Yaskawa INFORM job: R1_W27-A4(90,180)KM-OK.JBI

/JOB
//NAME R1_W27-A4(90,180)KM-OK
///FOLDERNAME KRIS-SCIANA
//POS
///NPOS 187,187,0,9,0,0
///TOOL 0
///POSTYPE PULSE
///PULSE
C00000=12408,-168229,-129239,-11856,76417,-1490
C00001=114075,-55562,-33330,-57879,69757,-51049
C00002=170127,-11218,4712,-80761,69619,-75034
C00003=166026,1115,14662,-80935,66751,-75417
C00004=166026,1115,14662,-80935,66751,-75417
C00005=164179,6139,17196,-85884,73779,-76491
C00006=163843,5639,16762,-85908,73539,-76507
C00007=164179,6139,17196,-85884,73779,-76491
C00008=166496,-467,13337,-75702,58764,-75189
C00009=166831,-1552,12436,-75705,58996,-75152
C00010=166508,-36,14521,-75997,58636,-74926
C00011=166831,-1552,12436,-75705,58996,-75152
C00012=166496,-467,13337,-75702,58764,-75189
C00013=166021,-3570,934,-78534,68009,-78358
C00014=137610,-28929,-19421,-69080,47942,-64710
C00015=100776,-35686,-23013,-57930,21837,-49720
C00016=103071,-36442,-26491,-56591,24205,-50318
C00017=97018,-28630,-27379,-22144,28331,-59500
C00018=96837,-21698,-21046,-22140,27966,-59499
C00019=100662,-29228,-19206,-55793,22319,-50751
C00020=102053,-30601,-20713,-56706,23278,-50281
C00021=94369,-26080,-26288,-14236,29524,-61616
C00022=90809,-41559,-31122,-11258,24098,-63096
C00023=90635,-42168,-31044,-11137,23721,-63156
C00024=94073,-53021,-44279,-15136,26788,-61156
C00025=105496,-45084,-28829,-64380,24182,-46446
C00026=105496,-45084,-28829,-64380,-61448,-46446
C00027=120732,-139011,-128731,-13191,-67324,37746
C00028=120732,-139011,-128731,-13191,-67324,37746
C00029=15630,-139011,-128731,-13191,-67324,37746
C00030=37783,65902,-41793,-18959,93512,79890
C00031=21816,-138429,-128213,-9073,25992,35710
C00032=3312,-138429,-128213,-9073,25992,35710
C00033=8567,85289,-13174,2735,78610,-10465
C00034=97991,22164,19578,-1121,74303,-36101
C00035=113962,41790,17661,4351,37010,-36101
C00036=153447,-77745,-45385,11807,63175,6285
C00037=169394,-84609,-38838,16107,56709,15659
C00038=173881,-75690,-28267,15647,54036,17014
C00039=174396,-73921,-25835,15662,53377,17117
C00040=174409,-72642,-23726,15788,52756,17025
C00041=174396,-73921,-25835,15662,53377,17117
C00042=177237,-69247,-20992,27235,53512,13633
C00043=177890,-67562,-19632,27129,53343,13864
C00044=177237,-69247,-20992,27235,53512,13633
C00045=181977,-77418,-24251,27266,50136,14704
C00046=193956,-50227,-14941,-539,58562,29056
C00047=192915,-50819,-15265,-329,58451,28665
C00048=194756,-48721,-14111,-700,58831,29355
C00049=182531,-71466,-31778,1788,58094,24759
C00050=122199,17749,55230,64618,69888,-3761
C00051=124469,25360,65490,65961,67496,-4502
C00052=125352,28797,70143,66592,66515,-4877
C00053=125200,39134,82378,67427,65683,-5911
C00054=125978,39297,82548,67654,65232,-5820
C00055=125200,39134,82378,67427,65683,-5911
C00056=125352,28797,70143,66592,66515,-4877
C00057=127676,20892,69191,78285,59026,-9362
C00058=127562,25294,74286,78756,58894,-9826
C00059=127676,21375,69995,78428,58968,-9490
C00060=125009,20842,69444,77518,60577,-9664
C00061=122672,36678,78518,58027,73309,-3381
C00062=122677,38905,82216,58303,72687,-3837
C00063=122672,36678,78518,58027,73309,-3381
C00064=169394,-84609,-38838,16107,56709,15659
C00065=192177,-39033,-19160,299,85673,46850
C00066=192177,-34142,-7713,300,81140,46844
C00067=191273,-36033,-8917,230,80912,46543
C00068=190571,-37450,-9806,174,80732,46307
C00069=191000,-36591,-9270,208,80842,46449
C00070=191000,-37231,-10676,208,81378,46450
C00071=190373,-38486,-11456,158,81216,46242
C00072=190373,-38091,-10592,158,80886,46242
C00073=190373,-40536,-16053,159,82992,46244
C00074=118612,15198,38856,55022,83195,1057
C00075=133487,-1087,21013,35992,98849,64323
C00076=137132,-5726,26455,36615,92702,63739
C00077=137287,-7082,25375,36660,92613,63770
C00078=137132,-5726,26455,36615,92702,63739
C00079=137132,-4574,28724,36576,92049,63519
C00080=137132,-5726,26455,36615,92702,63739
C00081=135105,9364,31394,36359,97356,64485
C00082=137553,-19599,1652,32898,84560,61916
C00083=145396,-31747,-6442,33707,80478,63803
C00084=146058,-32230,-6758,33764,80175,63976
C00085=145396,-31747,-6442,33707,80478,63803
C00086=145396,-32381,-7876,33664,80944,63945
C00087=145635,-34810,-9443,33705,80615,63940
C00088=145635,-34478,-8700,33728,80373,63868
C00089=145635,-34810,-9443,33705,80615,63940
C00090=166958,-28260,-6522,34091,73535,70390
C00091=170921,-25100,-2173,34137,71094,71258
C00092=171490,-25282,-2297,34116,70859,71419
C00093=170921,-25100,-2173,34137,71094,71258
C00094=170921,-25785,-3769,34024,71622,71427
C00095=171866,-27898,-5215,34016,71085,71649
C00096=171866,-27525,-4348,34079,70800,71557
C00097=171866,-27898,-5215,34016,71085,71649
C00098=170413,-50683,-19184,37966,51947,77320
C00099=172186,-18361,1190,35695,54496,79271
C00100=175964,-9154,13477,35828,50627,79612
C00101=176352,-9219,13425,35709,50467,79746
C00102=175964,-9154,13477,35828,50627,79612
C00103=175964,-10038,11459,35461,51274,79877
C00104=176713,-11464,10718,35354,50747,80043
C00105=176713,-11144,11450,35487,50511,79947
C00106=176713,-11464,10718,35354,50747,80043
C00107=123076,-83185,-29574,44713,66004,60586
C00108=132807,-78951,-22653,44198,75112,68451
C00109=133029,-79369,-22050,44355,74587,68307
C00110=133442,-81220,-22681,44553,73994,68215
C00111=133280,-79395,-22588,44357,74706,68467
C00112=133284,-82173,-24950,44353,74724,68477
C00113=133854,-84143,-25057,44659,73784,68294
C00114=133789,-83559,-24494,44652,73780,68264
C00115=133789,-82965,-23605,44700,73605,68182
C00116=133789,-83559,-24494,44652,73780,68264
C00117=126764,-78223,-26799,42400,79954,67989
C00118=129779,-124310,-39885,59101,44128,50595
C00119=142359,-111009,-28991,70365,32429,46878
C00120=144435,-110863,-28981,70591,31368,47293
C00121=166637,-108168,-28907,68791,20141,53479
C00122=165685,-116661,-37003,67388,20889,53934
C00123=169317,-97643,-42504,39636,61921,25134
C00124=181806,-47831,-14195,30226,94440,40482
C00125=192217,-74733,-34955,23643,74815,40848
C00126=189039,-36338,-14362,23914,80418,40542
C00127=179036,-43494,-16720,35248,78492,35239
C00128=184921,-32781,-12708,31409,62196,49986
C00129=184567,-29470,-5587,32219,59878,49253
C00130=185969,-1035,16805,31607,54976,48516
C00131=184454,-6788,8530,31302,57322,48585
C00132=186295,-45172,-18023,32156,53759,48198
C00133=187719,-75788,-33082,34439,47747,46698
C00134=196206,-71365,-30868,20961,47500,52163
C00135=191632,-40680,-12057,24621,48037,49834
C00136=186300,-39428,-14940,31590,54648,48556
C00137=172329,-61780,-29172,35843,57798,43133
C00138=136853,-81161,-37735,39391,69197,31515
C00139=139314,-24647,17192,44556,110664,42025
C00140=134198,-53539,2603,44314,98424,40161
C00141=147007,-50232,4151,49976,93054,43060
C00142=144010,-50727,1445,48871,95437,42954
C00143=139156,-48548,-22547,50335,108120,47151
C00144=122197,265,20116,61362,75919,1585
C00145=148312,-18266,18073,35868,41105,22148
C00146=148389,-10811,27499,37215,39474,21366
C00147=148139,-7130,31782,37859,38978,20950
C00148=149047,-9416,30148,37653,38478,21229
C00149=148550,-6621,33826,38481,38019,20665
C00150=151250,-3570,34403,36506,37914,22272
C00151=150396,-8469,29288,36370,38763,22201
C00152=150383,-15985,19712,34952,40435,23027
C00153=136141,-317,34070,49048,57432,19039
C00154=137229,7022,44527,50381,55121,18205
C00155=137621,10190,48745,50908,54295,17886
C00156=137107,11277,51332,51470,53891,17317
C00157=136657,9562,48504,50983,54669,17581
C00158=137398,10846,49256,50891,54423,17845
C00159=137247,10896,49257,50876,54513,17818
C00160=136822,13685,51719,50910,54678,17683
C00161=136799,9316,46568,50416,55288,18069
C00162=135467,4556,38210,49073,57743,18855
C00163=136137,-10257,13643,45943,62583,21899
C00164=136139,-13457,6254,44950,64655,-57340
C00165=140525,19486,41917,27486,58532,-69458
C00166=158575,-22743,-5640,261,63822,-52267
C00167=201270,-72526,-20170,-41599,43995,-22865
C00168=208523,-61328,-5512,-45049,45103,-18922
C00169=210983,-54521,-945,-44398,50079,-19814
C00170=208926,-60351,-4855,-45020,45353,-18846
C00171=208139,-60468,-3279,-45679,44265,-18612
C00172=209884,-54474,-922,-44345,49597,-20126
C00173=202908,-51930,157,-43430,46646,-22304
C00174=208516,-61339,-5515,-45051,45097,-18922
C00175=207445,-70087,-17224,-43111,46602,-20424
C00176=181249,-65588,-30997,1667,65478,-39835
C00177=185098,-71138,-35276,1207,65193,-38466
C00178=182759,-75971,-40143,1483,65742,61063
C00179=206355,-41348,-16857,-5174,86104,67834
C00180=205860,-39116,-9742,-5254,82857,67803
C00181=199217,-16106,8750,-10349,89886,65622
C00182=195049,-32120,-9942,-6453,85783,64063
C00183=178413,-64785,-35080,-8104,82994,58638
C00184=153142,-115476,-42163,-24127,19724,-41141
C00185=118343,-192417,-136241,31416,17665,-73466
C00186=12522,-192417,-136241,31416,17665,-73466
BC00000=5573,1179356,685508
BC00001=17842,1187216,744485
BC00002=145005,1191142,773938
BC00003=169645,1191142,773938
BC00004=169645,1191142,773938
BC00005=170825,1191142,715041
BC00006=170825,1191142,715041
BC00007=170825,1191142,715041
BC00008=193098,1191142,831231
BC00009=203526,1191142,830949
BC00010=203526,1191142,830949
BC00011=203526,1191142,830949
BC00012=193098,1191142,831231
BC00013=169645,1191142,773938
BC00014=112075,1191142,777374
BC00015=47018,1191142,781257
BC00016=50087,1191142,764866
BC00017=51351,1191141,771759
BC00018=51351,1191141,771759
BC00019=51315,1191142,758310
BC00020=51315,1191142,758310
BC00021=51315,1191142,758310
BC00022=51315,1191142,758310
BC00023=51315,1191142,758310
BC00024=51315,1191142,758310
BC00025=47056,1191142,794711
BC00026=20889,1191142,794711
BC00027=33296,1190075,947302
BC00028=33296,691954,947302
BC00029=33296,691954,947302
BC00030=150689,509,1059807
BC00031=165933,1190075,1065356
BC00032=165933,1346249,1065356
BC00033=73688,729726,969252
BC00034=389559,778302,1060448
BC00035=389559,1189504,1060448
BC00036=393628,1104806,555119
BC00037=394257,1091704,476953
BC00038=399035,1282079,493083
BC00039=399035,1280810,493083
BC00040=399035,1280810,493083
BC00041=399035,1280810,493083
BC00042=399035,1261438,493083
BC00043=399035,1261313,493083
BC00044=399035,1261438,493083
BC00045=399035,1261438,493083
BC00046=399035,1290178,493083
BC00047=399035,1288101,493083
BC00048=399035,1290178,493083
BC00049=399035,1296613,493602
BC00050=399035,1384690,493083
BC00051=399035,1384690,493083
BC00052=399035,1384690,493083
BC00053=399035,1382924,493083
BC00054=399035,1382921,493083
BC00055=399035,1382924,493083
BC00056=399035,1384690,493083
BC00057=399035,1384690,493083
BC00058=399035,1384690,493083
BC00059=399035,1384690,493083
BC00060=399035,1384690,493083
BC00061=399035,1366830,493083
BC00062=399035,1367204,493083
BC00063=399035,1366830,493083
BC00064=394257,1091704,476953
BC00065=394257,1091704,476953
BC00066=394257,1091704,476953
BC00067=394257,1091704,476953
BC00068=394257,1091704,476953
BC00069=394257,1091704,476953
BC00070=394257,1091704,476953
BC00071=394257,1091704,476953
BC00072=394257,1091704,476953
BC00073=394257,1091704,476953
BC00074=394257,1176346,476953
BC00075=394257,1176346,476953
BC00076=394257,1176346,476953
BC00077=394257,1176346,476953
BC00078=394257,1176346,476953
BC00079=394257,1176346,476953
BC00080=394257,1176346,476953
BC00081=394257,1176346,476952
BC00082=394257,1176346,875295
BC00083=394257,1176346,875295
BC00084=394257,1176346,875295
BC00085=394257,1176346,875295
BC00086=394257,1176346,875295
BC00087=394257,1176346,875295
BC00088=394257,1176346,875295
BC00089=394257,1176346,875295
BC00090=394257,1118001,875294
BC00091=394257,1118001,875294
BC00092=394257,1118001,875294
BC00093=394257,1118001,875294
BC00094=394257,1118001,875294
BC00095=394257,1118001,875294
BC00096=394257,1118001,875294
BC00097=394257,1118001,875294
BC00098=394257,1118001,875294
BC00099=394257,1118001,875294
BC00100=394257,1118001,875294
BC00101=394257,1118001,875294
BC00102=394257,1118001,875294
BC00103=394257,1118001,875294
BC00104=394257,1118001,875294
BC00105=394257,1118001,875294
BC00106=394257,1118001,875294
BC00107=394257,1118001,875294
BC00108=394257,1118001,875294
BC00109=394257,1118001,875294
BC00110=394257,1118001,875294
BC00111=394257,1118001,875294
BC00112=394257,1118001,875294
BC00113=394257,1118001,875294
BC00114=394257,1118001,875294
BC00115=394257,1118001,875294
BC00116=394257,1118001,875294
BC00117=394257,1118001,875294
BC00118=394257,1118001,875294
BC00119=394257,1138852,875294
BC00120=394257,1138852,875294
BC00121=394257,1138852,875294
BC00122=394257,1138852,875294
BC00123=394257,1101222,875294
BC00124=394257,1101222,875294
BC00125=394257,1101222,875294
BC00126=394257,1101222,875294
BC00127=394257,1101222,875294
BC00128=394257,1101222,875292
BC00129=394257,1101222,875294
BC00130=394257,1101222,875294
BC00131=394257,1101222,875294
BC00132=394257,1101222,875294
BC00133=394257,1101222,875294
BC00134=394257,1101222,875294
BC00135=394257,1101222,875294
BC00136=394257,1101222,875294
BC00137=394257,1101222,875294
BC00138=394257,1101222,875294
BC00139=394257,1101222,444692
BC00140=394257,1101222,444692
BC00141=394257,1101222,444692
BC00142=394257,1101222,444692
BC00143=394257,1102104,444737
BC00144=399035,1384690,465371
BC00145=399035,1384690,493083
BC00146=399035,1384690,493083
BC00147=399035,1384690,493083
BC00148=399035,1384690,493083
BC00149=399035,1384690,493083
BC00150=399035,1384690,493083
BC00151=399035,1384690,493083
BC00152=399035,1384690,493083
BC00153=399035,1384690,493083
BC00154=399035,1384690,493083
BC00155=399035,1384690,493083
BC00156=399035,1384690,493083
BC00157=399035,1384690,493083
BC00158=399035,1384690,493083
BC00159=399035,1381411,493083
BC00160=399035,1380262,493083
BC00161=399035,1381408,493083
BC00162=399035,1384272,493083
BC00163=399035,1384690,482138
BC00164=399035,1384690,452684
BC00165=399035,1384690,493083
BC00166=399035,1345582,493083
BC00167=399035,1287971,493083
BC00168=399035,1285341,493083
BC00169=399035,1284289,493083
BC00170=399035,1284289,493083
BC00171=399035,1284289,493083
BC00172=399035,1284289,493083
BC00173=399035,1284289,493083
BC00174=399035,1274155,493083
BC00175=399035,1276785,493083
BC00176=399035,1276785,493083
BC00177=399035,1276785,493083
BC00178=394257,1083237,476953
BC00179=394257,1083237,476953
BC00180=394257,1083237,476953
BC00181=394257,1083237,476953
BC00182=394257,1083237,476953
BC00183=394257,1083237,476953
BC00184=394257,1083237,476953
BC00185=394257,908728,1014252
BC00186=189642,706603,1014252
///POSTYPE BASE
///RECTAN
///RCONF 0,0,0,0,0,0,0,0,0,0,0,0,0,0,0,0,0,0,0,0,0,0,0,0
P00006=0.222,-3.123,-1.508,0.0000,0.0000,0.0000
P00021=-0.225,-6.128,-0.405,0.0000,0.0000,0.0000
P00022=0.222,-3.123,-1.508,0.0000,0.0000,0.0000
P00023=0.143,-0.036,0.682,0.0000,0.0000,0.0000
P00024=0.145,-0.552,1.326,0.0000,0.0000,0.0000
P00025=-2.003,0.006,0.728,0.0000,0.0000,0.0000
P00026=0.562,-0.002,-0.337,0.0000,0.0000,0.0000
P00027=-0.746,0.015,-9.096,0.0000,0.0000,0.0000
P00050=4.296,-4.501,-0.826,0.0000,0.0000,0.0000
//INST
///DATE 2024/07/30 11:30
///ATTR SC,RW
///GROUP1 RB1,BS1
NOP
'r1_W27-A4(90,180)
'Path S1000
SFTOF
MOVJ C00000 BC00000 VJ=100.00
MOVJ C00001 BC00001 VJ=100.00
MOVJ C00002 BC00002 VJ=100.00
MOVJ C00003 BC00003 VJ=100.00
MOVL C00004 BC00004 V=166.7
MOVL C00005 BC00005 V=60.0
REFP 3 C00006 BC00006
CALL JOB:SEARCH-R1
SET P023 P006
SFTON P023
MOVL C00007 BC00007 V=60.0
MOVL C00008 BC00008 V=100.0
MOVL C00009 BC00009 V=60.0
REFP 3 C00010 BC00010
CALL JOB:SEARCH-R1
SET P023 P006
SFTON P023
MOVL C00011 BC00011 V=60.0
MOVL C00012 BC00012 V=100.0
'Path VIA1106
SFTOF
MOVJ C00013 BC00013 VJ=20.00
'Path W1001
SFTOF
SFTON P023
MOVJ C00014 BC00014 VJ=20.00
MOVJ C00015 BC00015 VJ=20.00
MOVJ C00016 BC00016 VJ=20.00
MOVL C00017 BC00017 V=166.7 PL=0
MOVL C00018 BC00018 V=166.7
REFP 1 C00019 BC00019
REFP 2 C00020 BC00020
MACRO1 MJ#(0) ARGF7
ARCON
MOVL C00021 BC00021 V=10.8
MOVL C00022 BC00022 V=10.8
MOVL C00023 BC00023 V=10.8
ARCOF
MOVL C00024 BC00024 V=166.7
MOVL C00025 BC00025 V=166.7
SFTOF
'Path VIA1107
SFTOF
MOVJ C00026 BC00026 VJ=40.00
'Path VIA1103
SFTOF
MOVJ C00027 BC00027 VJ=100.00
MOVJ C00028 BC00028 VJ=100.00
MOVJ C00029 BC00029 VJ=100.00
COMM MOVJ C00030 BC00030 VJ=100.00
'Path VIA1104
SFTOF
COMM MOVJ C00031 BC00031 VJ=60.00
COMM MOVJ C00032 BC00032 VJ=30.00
'Path VIA1105
SFTOF
CALL JOB:ONLY_CUT_KM_NEW_SCIANA
MOVJ C00033 BC00033 VJ=100.00
MOVJ C00034 BC00034 VJ=100.00
MOVJ C00035 BC00035 VJ=60.00
SFTOF
MOVJ C00036 BC00036 VJ=80.00
MOVL C00037 BC00037 V=250.0
COMM PAUSE
COMM MOVL C00038 BC00038 V=166.7
COMM MOVL C00039 BC00039 V=60.0
COMM REFP 3 C00040 BC00040
COMM CALL JOB:SEARCH-R1
COMM SET P026 P006
COMM SFTON P026
COMM MOVL C00041 BC00041 V=60.0
COMM MOVL C00042 BC00042 V=60.0
COMM REFP 3 C00043 BC00043
COMM CALL JOB:SEARCH-R1
COMM SET P026 P006
COMM SFTON P026
COMM MOVL C00044 BC00044 V=60.0
COMM MOVL C00045 BC00045 V=100.0
COMM MOVL C00046 BC00046 V=60.0
COMM REFP 3 C00047 BC00047
COMM CALL JOB:SEARCH-R1
COMM SET P026 P006
COMM SFTON P026
COMM MOVL C00048 BC00048 V=60.0
COMM MOVL C00049 BC00049 V=166.7
COMM 'Path S1004
COMM SFTOF
COMM MOVL C00050 BC00050 V=166.7
COMM MOVL C00051 BC00051 V=166.7
COMM MOVL C00052 BC00052 V=100.0
COMM MOVL C00053 BC00053 V=60.0
COMM REFP 3 C00054 BC00054
COMM CALL JOB:SEARCH-R1
COMM SET P027 P006
COMM SFTON P027
COMM MOVL C00055 BC00055 V=60.0
COMM MOVL C00056 BC00056 V=100.0
COMM MOVL C00057 BC00057 V=60.0
COMM REFP 3 C00058 BC00058
COMM CALL JOB:SEARCH-R1
COMM SET P027 P006
COMM SFTON P027
COMM MOVL C00059 BC00059 V=60.0
COMM MOVL C00060 BC00060 V=100.0
COMM MOVL C00061 BC00061 V=60.0
COMM REFP 3 C00062 BC00062
COMM CALL JOB:SEARCH-R1
COMM SET P027 P006
COMM SFTON P027
COMM MOVL C00063 BC00063 V=60.0
COMM PAUSE
MOVJ C00064 BC00064 VJ=100.00
'BP 060624
MOVL C00065 BC00065 V=250.0
MOVL C00066 BC00066 V=250.0
MOVL C00067 BC00067 V=166.7
REFP 3 C00068 BC00068
CALL JOB:SEARCH-R1
SET P050 P006
SFTON P050
MOVL C00069 BC00069 V=60.0
MOVL C00070 BC00070 V=100.0
MOVL C00071 BC00071 V=60.0 PL=0
REFP 3 C00072 BC00072
CALL JOB:SEARCH-R1
SET P050 P006
SFTON P050
MOVL C00073 BC00073 V=60.0
SFTOF
MOVL C00074 BC00074 V=166.7
MOVJ C00075 BC00075 VJ=10.00
MOVL C00076 BC00076 V=66.7
REFP 3 C00077 BC00077
CALL JOB:SEARCH-R1
SET P021 P006
SFTON P021
MOVL C00078 BC00078 V=60.0
REFP 3 C00079 BC00079
CALL JOB:SEARCH-R1
SET P021 P006
SFTON P021
MOVL C00080 BC00080 V=60.0
MOVL C00081 BC00081 V=166.7
MOVL C00082 BC00082 V=250.0
MOVL C00083 BC00083 V=83.3
REFP 3 C00084 BC00084
CALL JOB:SEARCH-R1
SET P022 P006
SFTON P022
MOVL C00085 BC00085 V=60.0
MOVL C00086 BC00086 V=83.3
MOVL C00087 BC00087 V=83.3
REFP 3 C00088 BC00088
CALL JOB:SEARCH-R1
SET P022 P006
SFTON P022
MOVL C00089 BC00089 V=60.0
MOVL C00090 BC00090 V=166.7
SFTOF
MOVL C00091 BC00091 V=83.3
REFP 3 C00092 BC00092
CALL JOB:SEARCH-R1
SET P023 P006
SFTON P023
MOVL C00093 BC00093 V=100.0
MOVL C00094 BC00094 V=83.3
MOVL C00095 BC00095 V=100.0
REFP 3 C00096 BC00096
CALL JOB:SEARCH-R1
SET P023 P006
SFTON P023
MOVL C00097 BC00097 V=60.0
MOVL C00098 BC00098 V=100.0
MOVL C00099 BC00099 V=166.7
SFTOF
MOVL C00100 BC00100 V=166.7
REFP 3 C00101 BC00101
CALL JOB:SEARCH-R1
SET P024 P006
SFTON P024
MOVL C00102 BC00102 V=60.0
MOVL C00103 BC00103 V=83.3
MOVL C00104 BC00104 V=83.3
REFP 3 C00105 BC00105
CALL JOB:SEARCH-R1
SET P024 P006
SFTON P024
MOVL C00106 BC00106 V=60.0
MOVL C00107 BC00107 V=166.7
SFTOF
MOVL C00108 BC00108 V=166.7
MOVL C00109 BC00109 V=166.7
REFP 3 C00110 BC00110
CALL JOB:SEARCH-R1
SET P025 P006
SFTON P025
MOVL C00111 BC00111 V=60.0
MOVL C00112 BC00112 V=166.7
MOVL C00113 BC00113 V=166.7
MOVL C00114 BC00114 V=83.3
REFP 3 C00115 BC00115
CALL JOB:SEARCH-R1
SET P025 P006
SFTON P025
MOVL C00116 BC00116 V=60.0
SFTOF
MOVL C00117 BC00117 V=166.7
MOVL C00118 BC00118 V=166.7
SFTON P025
MACRO1 MJ#(0) ARGF6
MOVL C00119 BC00119 V=166.7
ARCON
MOVL C00120 BC00120 V=11.7
MOVL C00121 BC00121 V=11.7
ARCOF
SFTOF
MOVL C00122 BC00122 V=166.7
MOVL C00123 BC00123 V=166.7
SFTON P022
MACRO1 MJ#(0) ARGF7
MOVL C00124 BC00124 V=166.7 PL=0
ARCON
MOVL C00125 BC00125 V=11.7
MOVL C00126 BC00126 V=11.7
ARCOF
SFTOF
MOVJ C00127 BC00127 VJ=10.00
MOVJ C00128 BC00128 VJ=10.00
SFTON P024
MACRO1 MJ#(0) ARGF7
MOVJ C00129 BC00129 VJ=10.00
ARCON
MOVL C00130 BC00130 V=11.7
ARCOF
MOVJ C00131 BC00131 VJ=10.00
MOVJ C00132 BC00132 VJ=10.00
MOVJ C00133 BC00133 VJ=10.00
SFTOF
SFTOF
SFTON P023
MACRO1 MJ#(0) ARGF7
MOVJ C00134 BC00134 VJ=10.00 PL=0
ARCON
MOVL C00135 BC00135 V=11.7
ARCOF
MOVJ C00136 BC00136 VJ=10.00
SFTOF
MOVJ C00137 BC00137 VJ=10.00
MOVJ C00138 BC00138 VJ=10.00
MOVJ C00139 BC00139 VJ=20.00
SFTON P021
MACRO1 MJ#(0) ARGF7
MOVJ C00140 BC00140 VJ=15.00
ARCON
MOVL C00141 BC00141 V=9.2
ARCOF
MOVJ C00142 BC00142 VJ=10.00
MOVJ C00143 BC00143 VJ=100.00
COMM PAUSE
COMM 'SPAWANIE
COMM 'Path VIA1109
COMM SFTOF
COMM MOVJ C00144 BC00144 VJ=20.00
COMM 'Path W1005
COMM SFTOF
COMM SFTON P026
COMM MOVL C00145 BC00145 V=166.7
COMM MOVL C00146 BC00146 V=166.7
COMM 'COMMENT-SPR
COMM MOVL C00147 BC00147 V=100.0 PL=0
COMM REFP 1 C00148 BC00148
COMM REFP 2 C00149 BC00149
COMM MACRO1 MJ#(0) ARGF7
COMM MOVL C00150 BC00150 V=10.0
COMM ARCOF
COMM MOVL C00151 BC00151 V=166.7
COMM MOVL C00152 BC00152 V=166.7
COMM SFTOF
COMM 'Path W1006
COMM SFTOF
COMM SFTON P026
COMM MOVL C00153 BC00153 V=166.7
COMM MOVL C00154 BC00154 V=166.7
COMM MOVL C00155 BC00155 V=100.0 PL=0
COMM REFP 1 C00156 BC00156
COMM REFP 2 C00157 BC00157
COMM MACRO1 MJ#(0) ARGF7
COMM MOVL C00158 BC00158 V=11.0
COMM MOVL C00159 BC00159 V=11.0
COMM MOVL C00160 BC00160 V=11.0
COMM ARCOF
COMM MOVL C00161 BC00161 V=166.7
COMM MOVL C00162 BC00162 V=166.7
COMM SFTOF
COMM 'Path VIA1110
COMM SFTOF
COMM MOVJ C00163 BC00163 VJ=50.00
COMM 'Path VIA1111
COMM SFTOF
COMM MOVJ C00164 BC00164 VJ=50.00
COMM 'Path W1007
COMM SFTOF
COMM SFTON P026
COMM MOVL C00165 BC00165 V=166.7
COMM MOVJ C00166 BC00166 VJ=20.00
COMM SFTOF
COMM SFTON P027
COMM MOVL C00167 BC00167 V=166.7
COMM MOVL C00168 BC00168 V=166.7
COMM MOVL C00169 BC00169 V=100.0 PL=0
COMM REFP 1 C00170 BC00170
COMM REFP 2 C00171 BC00171
COMM MACRO1 MJ#(0) ARGF9
COMM ARCON
COMM MOVL C00172 BC00172 V=6.7
COMM MOVL C00173 BC00173 V=6.7
COMM ARCOF
COMM MOVL C00174 BC00174 V=166.7
COMM MOVL C00175 BC00175 V=166.7
COMM SFTOF
COMM MOVL C00176 BC00176 V=166.7
COMM MOVJ C00177 BC00177 VJ=50.00
COMM PAUSE
MOVJ C00178 BC00178 VJ=50.00
MOVJ C00179 BC00179 VJ=50.00
SFTON P050
MACRO1 MJ#(0) ARGF7
MOVL C00180 BC00180 V=166.7 PL=0
ARCON
MOVL C00181 BC00181 V=10.8
ARCOF
MOVJ C00182 BC00182 VJ=15.00
SFTOF
MOVJ C00183 BC00183 VJ=50.00
MOVJ C00184 BC00184 VJ=100.00
MOVJ C00185 BC00185 VJ=100.00
MOVJ C00186 BC00186 VJ=50.00
END
